Staubli VAL3: get.pgx

public program get(string& x_sItem[] (dimensions=1), num x_nIndex (dimensions=1))
begin
end
